SYSTEM TEST_MATRIX (* Test IN_MATRIX with OUT_MATRIX *)
  (* Standard: 61499-1 *)
  (* Version 0.0, 2004-06-20, JHC, Rockwell Automation *)
  APPLICATION APP1
  END_APPLICATION
  DEVICE DEV1 : FRAME_DEVICE
    RESOURCE MATRICES : PANEL_RESOURCE
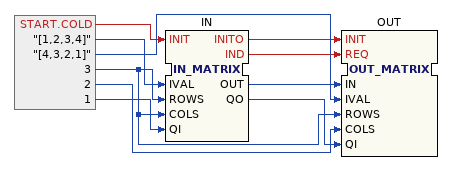
      FBS
        IN : IN_MATRIX;
        OUT : OUT_MATRIX;
      END_FBS
      EVENT_CONNECTIONS
        IN.INITO TO OUT.INIT;
        START.COLD TO IN.INIT;
        IN.IND TO OUT.REQ;
      END_CONNECTIONS
      DATA_CONNECTIONS
        IN.OUT TO OUT.IN;
        "[1,2,3,4]" TO IN.IVAL;
        "[4,3,2,1]" TO OUT.IVAL;
        3 TO IN.ROWS;
        3 TO IN.COLS;
        3 TO OUT.ROWS;
        2 TO OUT.COLS;
        1 TO IN.QI;
        IN.QO TO OUT.QI;
      END_CONNECTIONS
    END_RESOURCE
    DATA_CONNECTIONS
      1 TO MATRICES.ROWS;
      2 TO MATRICES.COLS;
    END_CONNECTIONS
  END_DEVICE
  DATA_CONNECTIONS (* parameter values *)
    [100,100,350,150] TO DEV1.BOUNDS;
    [1,1] TO DEV1.GRID;
  END_CONNECTIONS
END_SYSTEM
